(*
    Manual-mode interlock helper for maintenance positioning of DREAM DGPD.

    This function block assesses whether X, Y, and Z axes are all within a specified
    tolerance (fDelta) of their defined 'OUT' position. If so, bSafeToMoveRET is set TRUE,
    allowing safe movement of the RET axis (e.g., during maintenance or manual mode).
*)
FUNCTION_BLOCK FB_DGPDManual
VAR_IN_OUT
    astPositionStateX: ARRAY[1..GeneralConstants.MAX_STATES] OF ST_PositionState;
    astPositionStateY: ARRAY[1..GeneralConstants.MAX_STATES] OF ST_PositionState;
    astPositionStateZ: ARRAY[1..GeneralConstants.MAX_STATES] OF ST_PositionState;
    stMotionStageX: ST_MotionStage;
    stMotionStageY: ST_MotionStage;
    stMotionStageZ: ST_MotionStage;
END_VAR

VAR_OUTPUT
    bSafeToMoveRET: BOOL;            // TRUE if all axes are at OUT position within delta
END_VAR

IF NOT __ISVALIDREF(astPositionStateX)
    OR NOT __ISVALIDREF(astPositionStateY)
    OR NOT __ISVALIDREF(astPositionStateZ)
    OR NOT __ISVALIDREF(stMotionStageY)
    OR NOT __ISVALIDREF(stMotionStageZ)
    OR NOT __ISVALIDREF(stMotionStageX )
THEN
    RETURN;
END_IF

// --- Maintenance Mode RET Move Interlock Logic ---
bSafeToMoveRET := TRUE;

// Only when all are within tolerance, RET is safe to move
bSafeToMoveRET := ABS(stMotionStageX.Axis.NcToPlc.ActPos - astPositionStateX[E_DGPDState.OUT].fPosition) <= astPositionStateX[E_DGPDState.OUT].fDelta
                  AND  ABS(stMotionStageY.Axis.NcToPlc.ActPos - astPositionStateY[E_DGPDState.OUT].fPosition) <= astPositionStateY[E_DGPDState.OUT].fDelta
                  AND  ABS(stMotionStageZ.Axis.NcToPlc.ActPos - astPositionStateZ[E_DGPDState.OUT].fPosition) <= astPositionStateZ[E_DGPDState.OUT].fDelta;

END_FUNCTION_BLOCK

(* stored: Version 1.1.0.1
   POU FB_DGPDManual: Id {39ae7374-d9aa-4e7c-96db-2f110a50d3fa}, SpecialFunc None *)
